{attribute 'qualified_only'}
{attribute 'strict'}
TYPE OrderToteCommand:
(
DO_NOTHING	:=0,
LOAD		:=1,
UNLOAD		:=2,
SWAP		:=3,
OPEN_BAG	:=4,
STOP		:=5
);
END_TYPE

(* stored: Version 1.1.0.1, ProductVersion 3.1.4024.12
   DUT OrderToteCommand: Id {f0996174-fba0-4acd-aba5-f4f53a64f01f} *)
